// TIA Portal V16 export
// export: Created 2022-11-14T17:35:17.0009198Z, ExportSetting WithDefaults, DisplayName Totally Integrated Automation Portal, DisplayVersion V16, DisplayName TIA Portal Version Control Interface, DisplayVersion V16, DisplayName TIA Portal Openness, DisplayVersion V16, DisplayName STEP 7 Professional, DisplayVersion V16, DisplayName STEP 7 Safety, DisplayVersion V16, DisplayName WinCC Advanced, DisplayVersion V16
FUNCTION "FC03_TechnoplatAux" : Void   // FC3, LAD
TITLE = Auxiliary memory for the machine
{ S7_Optimized_Access := 'FALSE' }
AUTHOR : Robopac
VERSION : 0.0
// stored: AutoNumber false, IsIECCheckEnabled false, SetENOAutomatically false, UDAEnableTagReadback false
   VAR_INPUT
      PHASE : Bool;
   END_VAR
   VAR_TEMP
      Pulse_Reset : Bool;   // Pulse to reset encoders
      SuppSpeed : DWord;
      TempInt_min : Int;
      TempInt_max : Int;
      TempDint : DInt;
   END_VAR
   VAR_TEMP   // added for the SCL form of the ladder/FBD networks
      _w1 : Bool;
      _w2 : Bool;
      _w3 : Bool;
      _w4 : Bool;
   END_VAR
BEGIN

REGION Network 1: OSR and OSF for table phases sensor
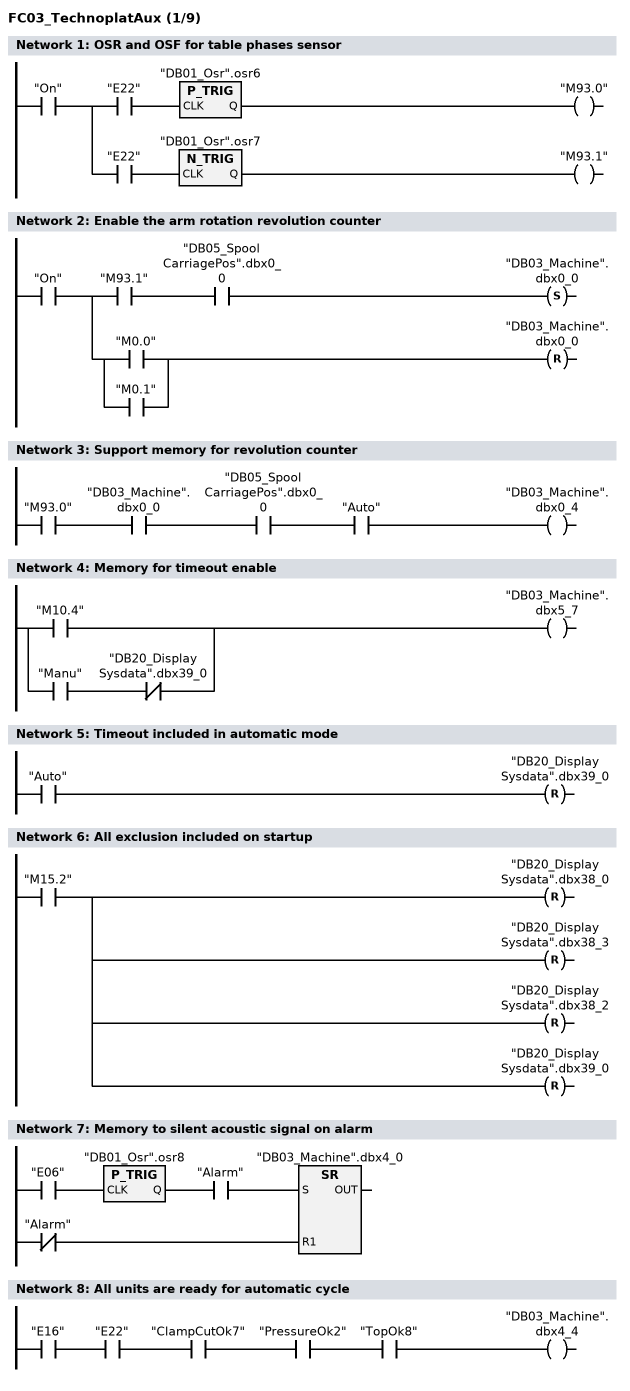
   RUNG wire#powerrail
      Contact( "On" )
      wire#w1
      Contact( "E22" )
      P_Trig( "DB01_Osr".osr6 )
      Coil( "M93.0" )
   END_RUNG
   RUNG wire#w1
      Contact( "E22" )
      N_Trig( "DB01_Osr".osr7 )
      Coil( "M93.1" )
   END_RUNG
   // the same network as SCL:
   #_w1 := "On" AND "E22";
   #_w2 := #_w1 AND NOT "DB01_Osr".osr6;   // rising edge
   "DB01_Osr".osr6 := #_w1;
   "M93.0" := #_w2;
   #_w3 := "On" AND "E22";
   #_w4 := NOT #_w3 AND "DB01_Osr".osr7;   // falling edge
   "DB01_Osr".osr7 := #_w3;
   "M93.1" := #_w4;
END_REGION

REGION Network 2: Enable the arm rotation revolution counter
   RUNG wire#powerrail
      Contact( "On" )
      wire#w1
      Contact( "M93.1" )
      Contact( "DB05_SpoolCarriagePos".dbx0_0 )
      S_Coil( "DB03_Machine".dbx0_0 )
   END_RUNG
   RUNG wire#w1
      Contact( "M0.0" )
      wire#w2
      R_Coil( "DB03_Machine".dbx0_0 )
   END_RUNG
   RUNG wire#w1
      Contact( "M0.1" )
   END_RUNG wire#w2
   // the same network as SCL:
   IF "On" AND "M93.1" AND "DB05_SpoolCarriagePos".dbx0_0 THEN "DB03_Machine".dbx0_0 := TRUE; END_IF;
   IF "On" AND ("M0.0" OR "M0.1") THEN "DB03_Machine".dbx0_0 := FALSE; END_IF;
END_REGION

REGION Network 3: Support memory for revolution counter
   RUNG wire#powerrail
      Contact( "M93.0" )
      Contact( "DB03_Machine".dbx0_0 )
      Contact( "DB05_SpoolCarriagePos".dbx0_0 )
      Contact( "Auto" )
      Coil( "DB03_Machine".dbx0_4 )
   END_RUNG
   // the same network as SCL:
   "DB03_Machine".dbx0_4 := "M93.0" AND "DB03_Machine".dbx0_0 AND "DB05_SpoolCarriagePos".dbx0_0 AND "Auto";
END_REGION

REGION Network 4: Memory for timeout enable
   RUNG wire#powerrail
      Contact( "M10.4" )
      wire#w1
      Coil( "DB03_Machine".dbx5_7 )
   END_RUNG
   RUNG wire#powerrail
      Contact( "Manu" )
      I_Contact( "DB20_DisplaySysdata".dbx39_0 )
   END_RUNG wire#w1
   // the same network as SCL:
   "DB03_Machine".dbx5_7 := "M10.4" OR ("Manu" AND NOT "DB20_DisplaySysdata".dbx39_0);
END_REGION

REGION Network 5: Timeout included in automatic mode
   RUNG wire#powerrail
      Contact( "Auto" )
      R_Coil( "DB20_DisplaySysdata".dbx39_0 )
   END_RUNG
   // the same network as SCL:
   IF "Auto" THEN "DB20_DisplaySysdata".dbx39_0 := FALSE; END_IF;
END_REGION

REGION Network 6: All exclusion included on startup
   RUNG wire#powerrail
      Contact( "M15.2" )
      wire#w1
      R_Coil( "DB20_DisplaySysdata".dbx38_0 )
   END_RUNG
   RUNG wire#w1
      R_Coil( "DB20_DisplaySysdata".dbx38_3 )
   END_RUNG
   RUNG wire#w1
      R_Coil( "DB20_DisplaySysdata".dbx38_2 )
   END_RUNG
   RUNG wire#w1
      R_Coil( "DB20_DisplaySysdata".dbx39_0 )
   END_RUNG
   // the same network as SCL:
   IF "M15.2" THEN
       "DB20_DisplaySysdata".dbx38_0 := FALSE;
       "DB20_DisplaySysdata".dbx38_3 := FALSE;
       "DB20_DisplaySysdata".dbx38_2 := FALSE;
       "DB20_DisplaySysdata".dbx39_0 := FALSE;
   END_IF;
END_REGION

REGION Network 7: Memory to silent acoustic signal on alarm
   RUNG wire#powerrail
      Contact( "E06" )
      P_Trig( "DB01_Osr".osr8 )
      Contact( "Alarm" )
      S_SR(operand := "DB03_Machine".dbx4_0, r1 := wire#w1)
   END_RUNG
   RUNG wire#powerrail
      I_Contact( "Alarm" )
   END_RUNG wire#w1
   // the same network as SCL:
   #_w1 := "E06" AND NOT "DB01_Osr".osr8;   // rising edge
   "DB01_Osr".osr8 := "E06";
   IF #_w1 AND "Alarm" THEN
       "DB03_Machine".dbx4_0 := TRUE;   // SR flip-flop
   END_IF;
   IF NOT "Alarm" THEN "DB03_Machine".dbx4_0 := FALSE; END_IF;
END_REGION

REGION Network 8: All units are ready for automatic cycle
   RUNG wire#powerrail
      Contact( "E16" )
      Contact( "E22" )
      Contact( "ClampCutOk7" )
      Contact( "PressureOk2" )
      Contact( "TopOk8" )
      Coil( "DB03_Machine".dbx4_4 )
   END_RUNG
   // the same network as SCL:
   "DB03_Machine".dbx4_4 := "E16" AND "E22" AND "ClampCutOk7" AND "PressureOk2" AND "TopOk8";
END_REGION

REGION Network 9: Prearrangement automatic cycle
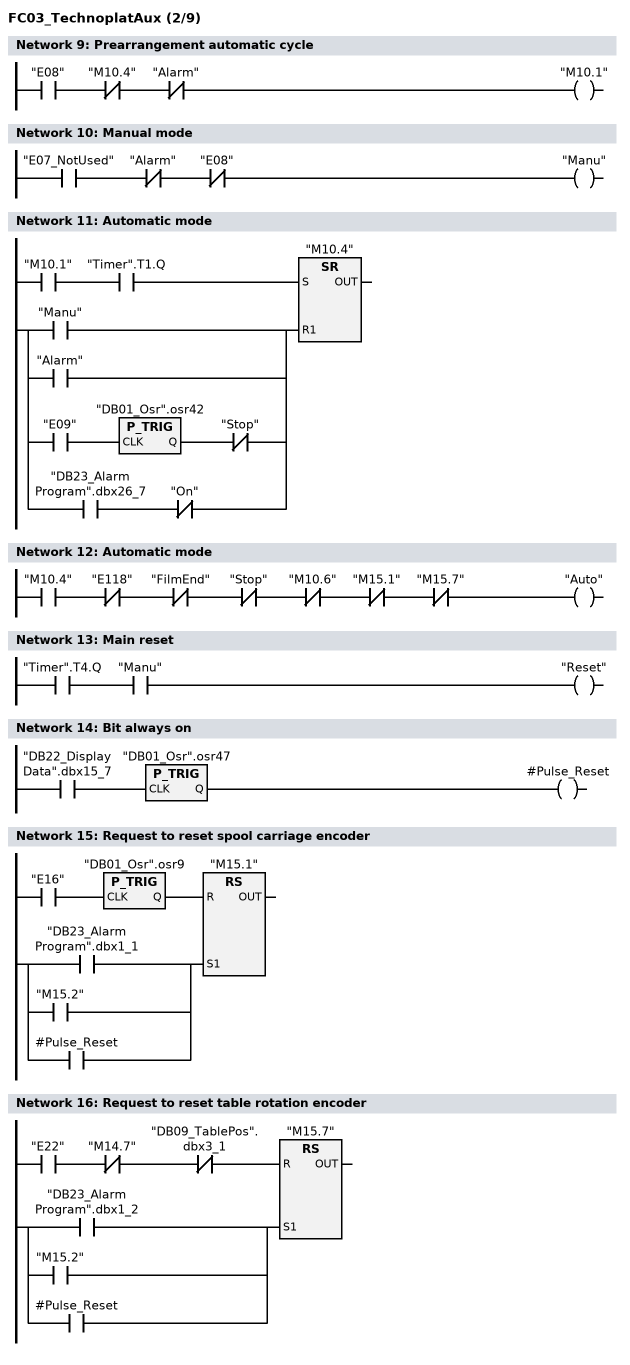
   RUNG wire#powerrail
      Contact( "E08" )
      I_Contact( "M10.4" )
      I_Contact( "Alarm" )
      Coil( "M10.1" )
   END_RUNG
   // the same network as SCL:
   "M10.1" := "E08" AND NOT "M10.4" AND NOT "Alarm";
END_REGION

REGION Network 10: Manual mode
   RUNG wire#powerrail
      Contact( "E07_NotUsed" )
      I_Contact( "Alarm" )
      I_Contact( "E08" )
      Coil( "Manu" )
   END_RUNG
   // the same network as SCL:
   "Manu" := "E07_NotUsed" AND NOT "Alarm" AND NOT "E08";
END_REGION

REGION Network 11: Automatic mode
   RUNG wire#powerrail
      Contact( "M10.1" )
      Contact( "Timer".T1.Q )
      S_SR(operand := "M10.4", r1 := wire#w1)
   END_RUNG
   RUNG wire#powerrail
      Contact( "Manu" )
   END_RUNG wire#w1
   RUNG wire#powerrail
      Contact( "Alarm" )
   END_RUNG wire#w1
   RUNG wire#powerrail
      Contact( "E09" )
      P_Trig( "DB01_Osr".osr42 )
      I_Contact( "Stop" )
   END_RUNG wire#w1
   RUNG wire#powerrail
      Contact( "DB23_AlarmProgram".dbx26_7 )
      I_Contact( "On" )
   END_RUNG wire#w1
   // the same network as SCL:
   #_w1 := "E09" AND NOT "DB01_Osr".osr42;   // rising edge
   "DB01_Osr".osr42 := "E09";
   IF "M10.1" AND "Timer".T1.Q THEN
       "M10.4" := TRUE;   // SR flip-flop
   END_IF;
   IF "Manu" OR "Alarm" OR (#_w1 AND NOT "Stop") OR ("DB23_AlarmProgram".dbx26_7 AND NOT "On") THEN
       "M10.4" := FALSE;
   END_IF;
END_REGION

REGION Network 12: Automatic mode
   RUNG wire#powerrail
      Contact( "M10.4" )
      I_Contact( "E118" )
      I_Contact( "FilmEnd" )
      I_Contact( "Stop" )
      I_Contact( "M10.6" )
      I_Contact( "M15.1" )
      I_Contact( "M15.7" )
      Coil( "Auto" )
   END_RUNG
   // the same network as SCL:
   "Auto" := "M10.4" AND NOT "E118" AND NOT "FilmEnd" AND NOT "Stop" AND NOT "M10.6" AND NOT "M15.1" AND NOT "M15.7";
END_REGION

REGION Network 13: Main reset
   RUNG wire#powerrail
      Contact( "Timer".T4.Q )
      Contact( "Manu" )
      Coil( "Reset" )
   END_RUNG
   // the same network as SCL:
   "Reset" := "Timer".T4.Q AND "Manu";
END_REGION

REGION Network 14: Bit always on
   RUNG wire#powerrail
      Contact( "DB22_DisplayData".dbx15_7 )
      P_Trig( "DB01_Osr".osr47 )
      Coil( #Pulse_Reset )
   END_RUNG
   // the same network as SCL:
   #_w1 := "DB22_DisplayData".dbx15_7 AND NOT "DB01_Osr".osr47;   // rising edge
   "DB01_Osr".osr47 := "DB22_DisplayData".dbx15_7;
   #Pulse_Reset := #_w1;
END_REGION

REGION Network 15: Request to reset spool carriage encoder
   RUNG wire#powerrail
      Contact( "E16" )
      P_Trig( "DB01_Osr".osr9 )
      S_RS(operand := "M15.1", s1 := wire#w1)
   END_RUNG
   RUNG wire#powerrail
      Contact( "DB23_AlarmProgram".dbx1_1 )
   END_RUNG wire#w1
   RUNG wire#powerrail
      Contact( "M15.2" )
   END_RUNG wire#w1
   RUNG wire#powerrail
      Contact( #Pulse_Reset )
   END_RUNG wire#w1
   // the same network as SCL:
   #_w1 := "E16" AND NOT "DB01_Osr".osr9;   // rising edge
   "DB01_Osr".osr9 := "E16";
   IF #_w1 THEN
       "M15.1" := FALSE;   // RS flip-flop
   END_IF;
   IF "DB23_AlarmProgram".dbx1_1 OR "M15.2" OR #Pulse_Reset THEN "M15.1" := TRUE; END_IF;
END_REGION

REGION Network 16: Request to reset table rotation encoder
   RUNG wire#powerrail
      Contact( "E22" )
      I_Contact( "M14.7" )
      I_Contact( "DB09_TablePos".dbx3_1 )
      S_RS(operand := "M15.7", s1 := wire#w1)
   END_RUNG
   RUNG wire#powerrail
      Contact( "DB23_AlarmProgram".dbx1_2 )
   END_RUNG wire#w1
   RUNG wire#powerrail
      Contact( "M15.2" )
   END_RUNG wire#w1
   RUNG wire#powerrail
      Contact( #Pulse_Reset )
   END_RUNG wire#w1
   // the same network as SCL:
   IF "E22" AND NOT "M14.7" AND NOT "DB09_TablePos".dbx3_1 THEN
       "M15.7" := FALSE;   // RS flip-flop
   END_IF;
   IF "DB23_AlarmProgram".dbx1_2 OR "M15.2" OR #Pulse_Reset THEN "M15.7" := TRUE; END_IF;
END_REGION

REGION Network 17: Table rotation backward to reset encoder
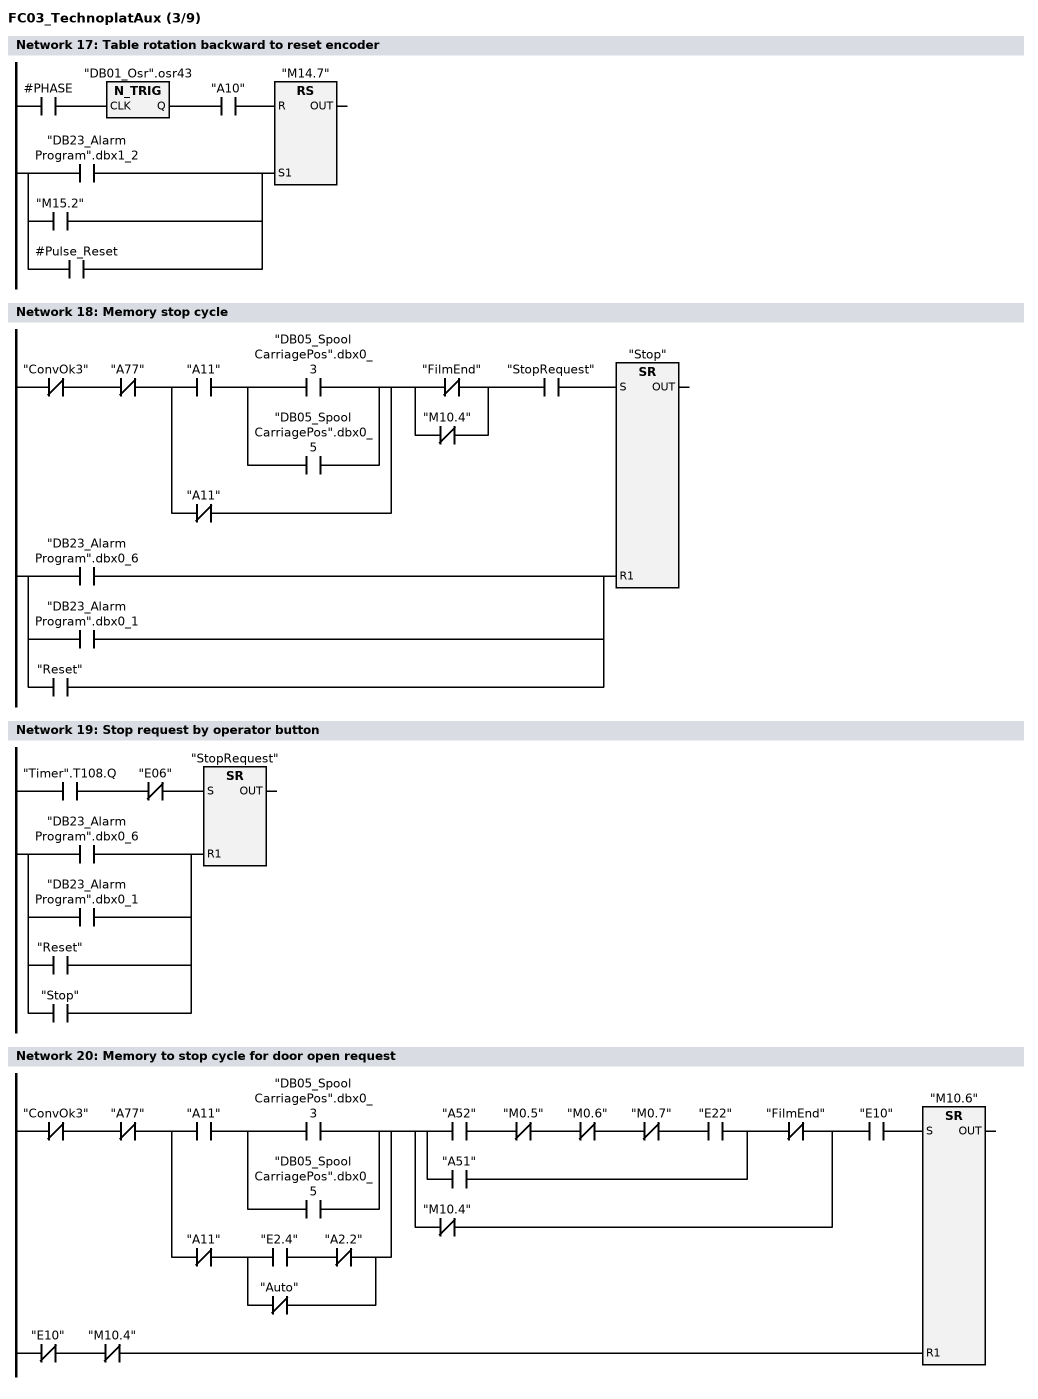
   RUNG wire#powerrail
      Contact( #PHASE )
      N_Trig( "DB01_Osr".osr43 )
      Contact( "A10" )
      S_RS(operand := "M14.7", s1 := wire#w1)
   END_RUNG
   RUNG wire#powerrail
      Contact( "DB23_AlarmProgram".dbx1_2 )
   END_RUNG wire#w1
   RUNG wire#powerrail
      Contact( "M15.2" )
   END_RUNG wire#w1
   RUNG wire#powerrail
      Contact( #Pulse_Reset )
   END_RUNG wire#w1
   // the same network as SCL:
   #_w1 := NOT #PHASE AND "DB01_Osr".osr43;   // falling edge
   "DB01_Osr".osr43 := #PHASE;
   IF #_w1 AND "A10" THEN
       "M14.7" := FALSE;   // RS flip-flop
   END_IF;
   IF "DB23_AlarmProgram".dbx1_2 OR "M15.2" OR #Pulse_Reset THEN "M14.7" := TRUE; END_IF;
END_REGION

REGION Network 18: Memory stop cycle
   RUNG wire#powerrail
      I_Contact( "ConvOk3" )
      I_Contact( "A77" )
      wire#w1
      Contact( "A11" )
      wire#w2
      Contact( "DB05_SpoolCarriagePos".dbx0_3 )
      wire#w3
      I_Contact( "FilmEnd" )
      wire#w4
      Contact( "StopRequest" )
      S_SR(operand := "Stop", r1 := wire#w5)
   END_RUNG
   RUNG wire#w2
      Contact( "DB05_SpoolCarriagePos".dbx0_5 )
   END_RUNG wire#w3
   RUNG wire#w1
      I_Contact( "A11" )
   END_RUNG wire#w3
   RUNG wire#w3
      I_Contact( "M10.4" )
   END_RUNG wire#w4
   RUNG wire#powerrail
      Contact( "DB23_AlarmProgram".dbx0_6 )
   END_RUNG wire#w5
   RUNG wire#powerrail
      Contact( "DB23_AlarmProgram".dbx0_1 )
   END_RUNG wire#w5
   RUNG wire#powerrail
      Contact( "Reset" )
   END_RUNG wire#w5
   // the same network as SCL:
   IF NOT "ConvOk3" AND NOT "A77" AND (("A11" AND ("DB05_SpoolCarriagePos".dbx0_3 OR "DB05_SpoolCarriagePos".dbx0_5)) OR NOT "A11") AND (NOT "FilmEnd" OR NOT "M10.4") AND "StopRequest" THEN
       "Stop" := TRUE;   // SR flip-flop
   END_IF;
   IF "DB23_AlarmProgram".dbx0_6 OR "DB23_AlarmProgram".dbx0_1 OR "Reset" THEN "Stop" := FALSE; END_IF;
END_REGION

REGION Network 19: Stop request by operator button
   RUNG wire#powerrail
      Contact( "Timer".T108.Q )
      I_Contact( "E06" )
      S_SR(operand := "StopRequest", r1 := wire#w1)
   END_RUNG
   RUNG wire#powerrail
      Contact( "DB23_AlarmProgram".dbx0_6 )
   END_RUNG wire#w1
   RUNG wire#powerrail
      Contact( "DB23_AlarmProgram".dbx0_1 )
   END_RUNG wire#w1
   RUNG wire#powerrail
      Contact( "Reset" )
   END_RUNG wire#w1
   RUNG wire#powerrail
      Contact( "Stop" )
   END_RUNG wire#w1
   // the same network as SCL:
   IF "Timer".T108.Q AND NOT "E06" THEN
       "StopRequest" := TRUE;   // SR flip-flop
   END_IF;
   IF "DB23_AlarmProgram".dbx0_6 OR "DB23_AlarmProgram".dbx0_1 OR "Reset" OR "Stop" THEN
       "StopRequest" := FALSE;
   END_IF;
END_REGION

REGION Network 20: Memory to stop cycle for door open request
   RUNG wire#powerrail
      I_Contact( "ConvOk3" )
      I_Contact( "A77" )
      wire#w1
      Contact( "A11" )
      wire#w2
      Contact( "DB05_SpoolCarriagePos".dbx0_3 )
      wire#w3
      Contact( "A52" )
      I_Contact( "M0.5" )
      I_Contact( "M0.6" )
      I_Contact( "M0.7" )
      Contact( "E22" )
      wire#w5
      I_Contact( "FilmEnd" )
      wire#w6
      Contact( "E10" )
      S_SR(operand := "M10.6", r1 := wire#w7)
   END_RUNG
   RUNG wire#w2
      Contact( "DB05_SpoolCarriagePos".dbx0_5 )
   END_RUNG wire#w3
   RUNG wire#w1
      I_Contact( "A11" )
      wire#w4
      Contact( "E2.4" )
      I_Contact( "A2.2" )
   END_RUNG wire#w3
   RUNG wire#w4
      I_Contact( "Auto" )
   END_RUNG wire#w3
   RUNG wire#w3
      Contact( "A51" )
   END_RUNG wire#w5
   RUNG wire#w3
      I_Contact( "M10.4" )
   END_RUNG wire#w6
   RUNG wire#powerrail
      I_Contact( "E10" )
      I_Contact( "M10.4" )
   END_RUNG wire#w7
   // the same network as SCL:
   IF NOT "ConvOk3" AND NOT "A77" AND (("A11" AND ("DB05_SpoolCarriagePos".dbx0_3 OR "DB05_SpoolCarriagePos".dbx0_5)) OR (NOT "A11" AND (("E2.4" AND NOT "A2.2") OR NOT "Auto"))) AND (((("A52" AND NOT "M0.5" AND NOT "M0.6" AND NOT "M0.7" AND "E22") OR "A51") AND NOT "FilmEnd") OR NOT "M10.4") AND "E10" THEN
       "M10.6" := TRUE;   // SR flip-flop
   END_IF;
   IF NOT "E10" AND NOT "M10.4" THEN "M10.6" := FALSE; END_IF;
END_REGION

REGION Network 21: Condition to check all out of positon alarm
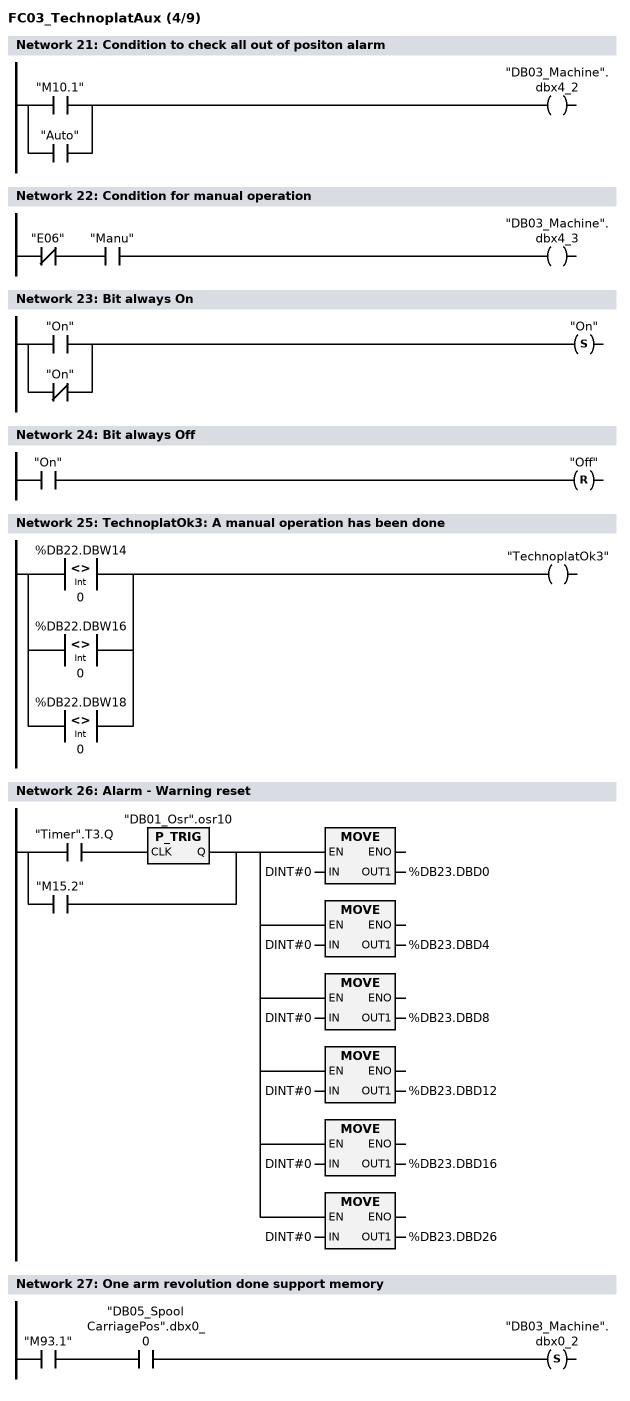
   RUNG wire#powerrail
      Contact( "M10.1" )
      wire#w1
      Coil( "DB03_Machine".dbx4_2 )
   END_RUNG
   RUNG wire#powerrail
      Contact( "Auto" )
   END_RUNG wire#w1
   // the same network as SCL:
   "DB03_Machine".dbx4_2 := "M10.1" OR "Auto";
END_REGION

REGION Network 22: Condition for manual operation
   RUNG wire#powerrail
      I_Contact( "E06" )
      Contact( "Manu" )
      Coil( "DB03_Machine".dbx4_3 )
   END_RUNG
   // the same network as SCL:
   "DB03_Machine".dbx4_3 := NOT "E06" AND "Manu";
END_REGION

REGION Network 23: Bit always On
   RUNG wire#powerrail
      Contact( "On" )
      wire#w1
      S_Coil( "On" )
   END_RUNG
   RUNG wire#powerrail
      I_Contact( "On" )
   END_RUNG wire#w1
   // the same network as SCL:
   IF "On" OR NOT "On" THEN "On" := TRUE; END_IF;
END_REGION

REGION Network 24: Bit always Off
   RUNG wire#powerrail
      Contact( "On" )
      R_Coil( "Off" )
   END_RUNG
   // the same network as SCL:
   IF "On" THEN "Off" := FALSE; END_IF;
END_REGION

REGION Network 25: TechnoplatOk3: A manual operation has been done
   RUNG wire#powerrail
      { S7_Templates := "SrcType := Int" } NE_Contact(in1 := %DB22.DBW14, in2 := 0)
      wire#w1
      Coil( "TechnoplatOk3" )
   END_RUNG
   RUNG wire#powerrail
      { S7_Templates := "SrcType := Int" } NE_Contact(in1 := %DB22.DBW16, in2 := 0)
   END_RUNG wire#w1
   RUNG wire#powerrail
      { S7_Templates := "SrcType := Int" } NE_Contact(in1 := %DB22.DBW18, in2 := 0)
   END_RUNG wire#w1
   // the same network as SCL:
   "TechnoplatOk3" := (%DB22.DBW14 <> 0) OR (%DB22.DBW16 <> 0) OR (%DB22.DBW18 <> 0);
END_REGION

REGION Network 26: Alarm - Warning reset
   RUNG wire#powerrail
      Contact( "Timer".T3.Q )
      P_Trig( "DB01_Osr".osr10 )
      wire#w1
      { S7_GenerateENO := "TRUE" } Move(in := DINT#0, out1 => %DB23.DBD0)
   END_RUNG
   RUNG wire#powerrail
      Contact( "M15.2" )
   END_RUNG wire#w1
   RUNG wire#w1
      { S7_GenerateENO := "TRUE" } Move(in := DINT#0, out1 => %DB23.DBD4)
   END_RUNG
   RUNG wire#w1
      { S7_GenerateENO := "TRUE" } Move(in := DINT#0, out1 => %DB23.DBD8)
   END_RUNG
   RUNG wire#w1
      { S7_GenerateENO := "TRUE" } Move(in := DINT#0, out1 => %DB23.DBD12)
   END_RUNG
   RUNG wire#w1
      { S7_GenerateENO := "TRUE" } Move(in := DINT#0, out1 => %DB23.DBD16)
   END_RUNG
   RUNG wire#w1
      { S7_GenerateENO := "TRUE" } Move(in := DINT#0, out1 => %DB23.DBD26)
   END_RUNG
   // the same network as SCL:
   #_w1 := "Timer".T3.Q AND NOT "DB01_Osr".osr10;   // rising edge
   "DB01_Osr".osr10 := "Timer".T3.Q;
   IF #_w1 OR "M15.2" THEN
       %DB23.DBD0 := DINT#0;
       %DB23.DBD4 := DINT#0;
       %DB23.DBD8 := DINT#0;
       %DB23.DBD12 := DINT#0;
       %DB23.DBD16 := DINT#0;
       %DB23.DBD26 := DINT#0;
   END_IF;
END_REGION

REGION Network 27: One arm revolution done support memory
   RUNG wire#powerrail
      Contact( "M93.1" )
      Contact( "DB05_SpoolCarriagePos".dbx0_0 )
      S_Coil( "DB03_Machine".dbx0_2 )
   END_RUNG
   // the same network as SCL:
   IF "M93.1" AND "DB05_SpoolCarriagePos".dbx0_0 THEN "DB03_Machine".dbx0_2 := TRUE; END_IF;
END_REGION

REGION Network 28: One arm revolution done
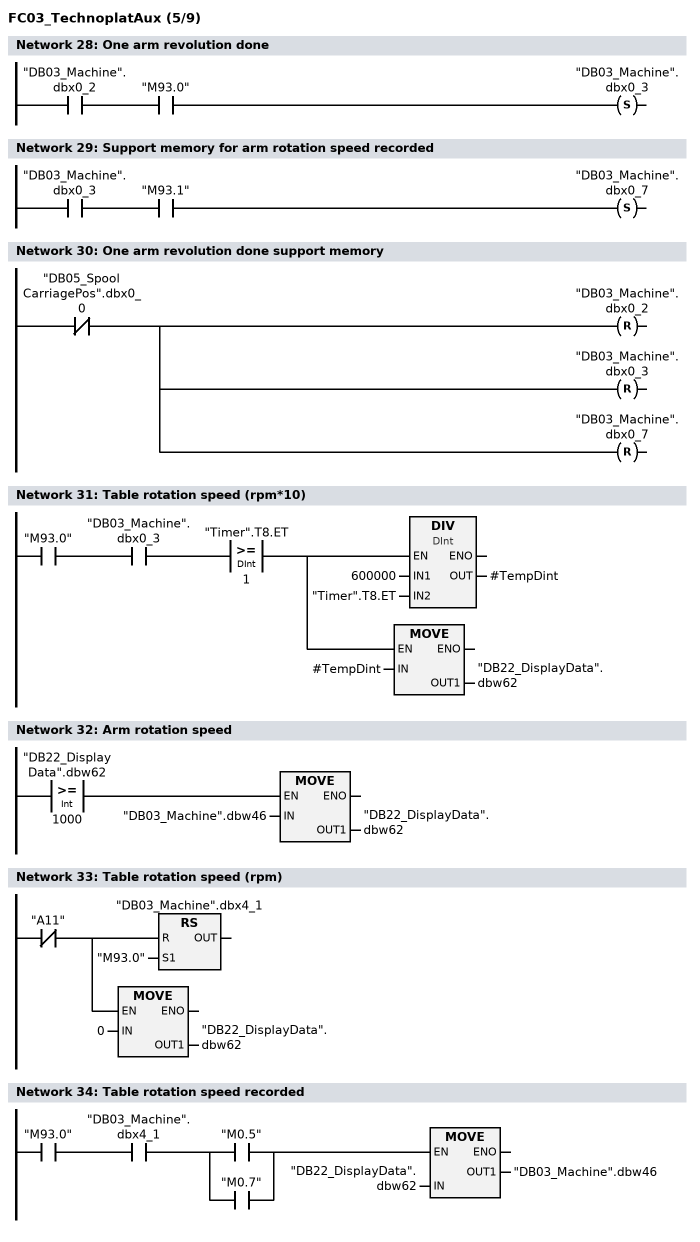
   RUNG wire#powerrail
      Contact( "DB03_Machine".dbx0_2 )
      Contact( "M93.0" )
      S_Coil( "DB03_Machine".dbx0_3 )
   END_RUNG
   // the same network as SCL:
   IF "DB03_Machine".dbx0_2 AND "M93.0" THEN "DB03_Machine".dbx0_3 := TRUE; END_IF;
END_REGION

REGION Network 29: Support memory for arm rotation speed recorded
   RUNG wire#powerrail
      Contact( "DB03_Machine".dbx0_3 )
      Contact( "M93.1" )
      S_Coil( "DB03_Machine".dbx0_7 )
   END_RUNG
   // the same network as SCL:
   IF "DB03_Machine".dbx0_3 AND "M93.1" THEN "DB03_Machine".dbx0_7 := TRUE; END_IF;
END_REGION

REGION Network 30: One arm revolution done support memory
   RUNG wire#powerrail
      I_Contact( "DB05_SpoolCarriagePos".dbx0_0 )
      wire#w1
      R_Coil( "DB03_Machine".dbx0_2 )
   END_RUNG
   RUNG wire#w1
      R_Coil( "DB03_Machine".dbx0_3 )
   END_RUNG
   RUNG wire#w1
      R_Coil( "DB03_Machine".dbx0_7 )
   END_RUNG
   // the same network as SCL:
   IF NOT "DB05_SpoolCarriagePos".dbx0_0 THEN
       "DB03_Machine".dbx0_2 := FALSE;
       "DB03_Machine".dbx0_3 := FALSE;
       "DB03_Machine".dbx0_7 := FALSE;
   END_IF;
END_REGION

REGION Network 31: Table rotation speed (rpm*10)
   RUNG wire#powerrail
      Contact( "M93.0" )
      Contact( "DB03_Machine".dbx0_3 )
      { S7_Templates := "SrcType := DInt" } GE_Contact(in1 := "Timer".T8.ET, in2 := 1)
      wire#w1
      { S7_Templates := "SrcType := DInt"; S7_GenerateENO := "TRUE" } Div(in1 := 600000, in2 := "Timer".T8.ET, out => #TempDint)
   END_RUNG
   RUNG wire#w1
      { S7_GenerateENO := "TRUE" } Move(in := #TempDint, out1 => "DB22_DisplayData".dbw62)
   END_RUNG
   // the same network as SCL:
   IF "M93.0" AND "DB03_Machine".dbx0_3 AND ("Timer".T8.ET >= 1) THEN
       #TempDint := 600000 / "Timer".T8.ET;
       "DB22_DisplayData".dbw62 := #TempDint;
   END_IF;
END_REGION

REGION Network 32: Arm rotation speed
   RUNG wire#powerrail
      { S7_Templates := "SrcType := Int" } GE_Contact(in1 := "DB22_DisplayData".dbw62, in2 := 1000)
      { S7_GenerateENO := "TRUE" } Move(in := "DB03_Machine".dbw46, out1 => "DB22_DisplayData".dbw62)
   END_RUNG
   // the same network as SCL:
   IF "DB22_DisplayData".dbw62 >= 1000 THEN "DB22_DisplayData".dbw62 := "DB03_Machine".dbw46; END_IF;
END_REGION

REGION Network 33: Table rotation speed (rpm)
   RUNG wire#powerrail
      I_Contact( "A11" )
      wire#w1
      S_RS(operand := "DB03_Machine".dbx4_1, s1 := "M93.0")
   END_RUNG
   RUNG wire#w1
      { S7_GenerateENO := "TRUE" } Move(in := 0, out1 => "DB22_DisplayData".dbw62)
   END_RUNG
   // the same network as SCL:
   IF NOT "A11" THEN
       "DB03_Machine".dbx4_1 := FALSE;   // RS flip-flop
   END_IF;
   IF "M93.0" THEN "DB03_Machine".dbx4_1 := TRUE; END_IF;
   IF NOT "A11" THEN "DB22_DisplayData".dbw62 := 0; END_IF;
END_REGION

REGION Network 34: Table rotation speed recorded
   RUNG wire#powerrail
      Contact( "M93.0" )
      Contact( "DB03_Machine".dbx4_1 )
      wire#w1
      Contact( "M0.5" )
      wire#w2
      { S7_GenerateENO := "TRUE" } Move(in := "DB22_DisplayData".dbw62, out1 => "DB03_Machine".dbw46)
   END_RUNG
   RUNG wire#w1
      Contact( "M0.7" )
   END_RUNG wire#w2
   // the same network as SCL:
   IF "M93.0" AND "DB03_Machine".dbx4_1 AND ("M0.5" OR "M0.7") THEN
       "DB03_Machine".dbw46 := "DB22_DisplayData".dbw62;
   END_IF;
END_REGION

REGION Network 35: Table rotation speed
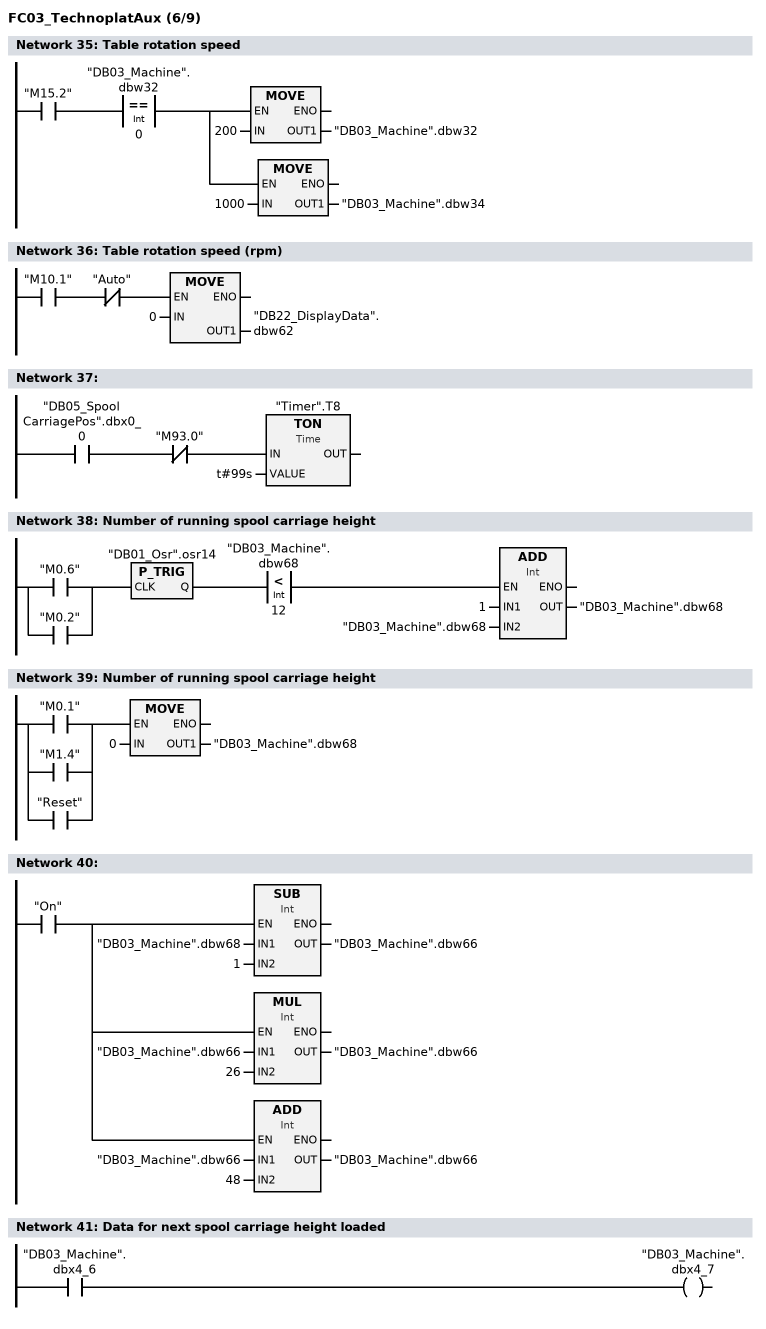
   RUNG wire#powerrail
      Contact( "M15.2" )
      { S7_Templates := "SrcType := Int" } EQ_Contact(in1 := "DB03_Machine".dbw32, in2 := 0)
      wire#w1
      { S7_GenerateENO := "TRUE" } Move(in := 200, out1 => "DB03_Machine".dbw32)
   END_RUNG
   RUNG wire#w1
      { S7_GenerateENO := "TRUE" } Move(in := 1000, out1 => "DB03_Machine".dbw34)
   END_RUNG
   // the same network as SCL:
   #_w1 := "M15.2" AND ("DB03_Machine".dbw32 = 0);
   IF #_w1 THEN
       "DB03_Machine".dbw32 := 200;
       "DB03_Machine".dbw34 := 1000;
   END_IF;
END_REGION

REGION Network 36: Table rotation speed (rpm)
   RUNG wire#powerrail
      Contact( "M10.1" )
      I_Contact( "Auto" )
      { S7_GenerateENO := "TRUE" } Move(in := 0, out1 => "DB22_DisplayData".dbw62)
   END_RUNG
   // the same network as SCL:
   IF "M10.1" AND NOT "Auto" THEN "DB22_DisplayData".dbw62 := 0; END_IF;
END_REGION

REGION Network 37
   "Timer".T8.TON(IN := "DB05_SpoolCarriagePos".dbx0_0 AND NOT "M93.0", PT := t#99s);   // TON coil
END_REGION

REGION Network 38: Number of running spool carriage height
   RUNG wire#powerrail
      Contact( "M0.6" )
      wire#w1
      P_Trig( "DB01_Osr".osr14 )
      { S7_Templates := "SrcType := Int" } LT_Contact(in1 := "DB03_Machine".dbw68, in2 := 12)
      { S7_Templates := "SrcType := Int"; S7_GenerateENO := "TRUE" } Add(in1 := 1, in2 := "DB03_Machine".dbw68, out => "DB03_Machine".dbw68)
   END_RUNG
   RUNG wire#powerrail
      Contact( "M0.2" )
   END_RUNG wire#w1
   // the same network as SCL:
   #_w1 := "M0.6" OR "M0.2";
   #_w2 := #_w1 AND NOT "DB01_Osr".osr14;   // rising edge
   "DB01_Osr".osr14 := #_w1;
   IF #_w2 AND ("DB03_Machine".dbw68 < 12) THEN "DB03_Machine".dbw68 := 1 + "DB03_Machine".dbw68; END_IF;
END_REGION

REGION Network 39: Number of running spool carriage height
   RUNG wire#powerrail
      Contact( "M0.1" )
      wire#w1
      { S7_GenerateENO := "TRUE" } Move(in := 0, out1 => "DB03_Machine".dbw68)
   END_RUNG
   RUNG wire#powerrail
      Contact( "M1.4" )
   END_RUNG wire#w1
   RUNG wire#powerrail
      Contact( "Reset" )
   END_RUNG wire#w1
   // the same network as SCL:
   IF "M0.1" OR "M1.4" OR "Reset" THEN "DB03_Machine".dbw68 := 0; END_IF;
END_REGION

REGION Network 40
   RUNG wire#powerrail
      Contact( "On" )
      wire#w1
      { S7_Templates := "SrcType := Int"; S7_GenerateENO := "TRUE" } Sub(in1 := "DB03_Machine".dbw68, in2 := 1, out => "DB03_Machine".dbw66)
   END_RUNG
   RUNG wire#w1
      { S7_Templates := "SrcType := Int"; S7_GenerateENO := "TRUE" } Mul(in1 := "DB03_Machine".dbw66, in2 := 26, out => "DB03_Machine".dbw66)
   END_RUNG
   RUNG wire#w1
      { S7_Templates := "SrcType := Int"; S7_GenerateENO := "TRUE" } Add(in1 := "DB03_Machine".dbw66, in2 := 48, out => "DB03_Machine".dbw66)
   END_RUNG
   // the same network as SCL:
   IF "On" THEN
       "DB03_Machine".dbw66 := "DB03_Machine".dbw68 - 1;
       "DB03_Machine".dbw66 := "DB03_Machine".dbw66 * 26;
       "DB03_Machine".dbw66 := "DB03_Machine".dbw66 + 48;
   END_IF;
END_REGION

REGION Network 41: Data for next spool carriage height loaded
   RUNG wire#powerrail
      Contact( "DB03_Machine".dbx4_6 )
      Coil( "DB03_Machine".dbx4_7 )
   END_RUNG
   // the same network as SCL:
   "DB03_Machine".dbx4_7 := "DB03_Machine".dbx4_6;
END_REGION

REGION Network 42: Moving data for the running quote
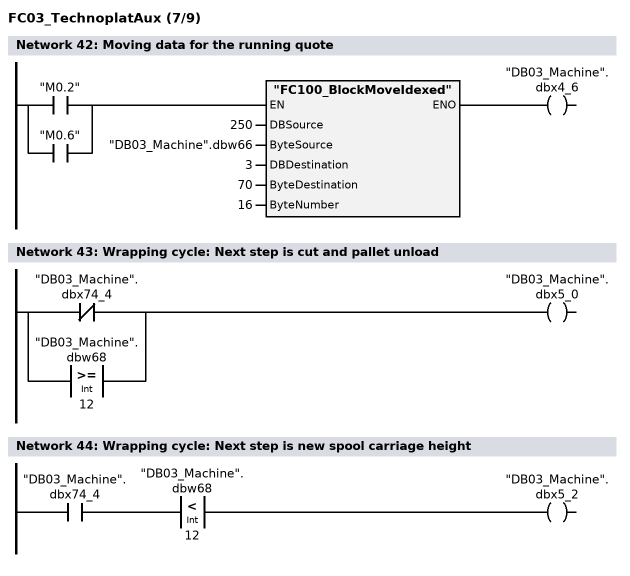
   RUNG wire#powerrail
      Contact( "M0.2" )
      wire#w1
      "FC100_BlockMoveIdexed"(DBSource := 250, ByteSource := "DB03_Machine".dbw66, DBDestination := 3, ByteDestination := 70, ByteNumber := 16)
      Coil( "DB03_Machine".dbx4_6 )
   END_RUNG
   RUNG wire#powerrail
      Contact( "M0.6" )
   END_RUNG wire#w1
   // the same network as SCL:
   "FC100_BlockMoveIdexed"(EN := "M0.2" OR "M0.6",
                           DBSource := 250,
                           ByteSource := "DB03_Machine".dbw66,
                           DBDestination := 3,
                           ByteDestination := 70,
                           ByteNumber := 16,
                           ENO => #_w1);
   "DB03_Machine".dbx4_6 := #_w1;
END_REGION

REGION Network 43: Wrapping cycle: Next step is cut and pallet unload
   RUNG wire#powerrail
      I_Contact( "DB03_Machine".dbx74_4 )
      wire#w1
      Coil( "DB03_Machine".dbx5_0 )
   END_RUNG
   RUNG wire#powerrail
      { S7_Templates := "SrcType := Int" } GE_Contact(in1 := "DB03_Machine".dbw68, in2 := 12)
   END_RUNG wire#w1
   // the same network as SCL:
   "DB03_Machine".dbx5_0 := NOT "DB03_Machine".dbx74_4 OR ("DB03_Machine".dbw68 >= 12);
END_REGION

REGION Network 44: Wrapping cycle: Next step is new spool carriage height
   RUNG wire#powerrail
      Contact( "DB03_Machine".dbx74_4 )
      { S7_Templates := "SrcType := Int" } LT_Contact(in1 := "DB03_Machine".dbw68, in2 := 12)
      Coil( "DB03_Machine".dbx5_2 )
   END_RUNG
   // the same network as SCL:
   "DB03_Machine".dbx5_2 := "DB03_Machine".dbx74_4 AND ("DB03_Machine".dbw68 < 12);
END_REGION

REGION Network 45: Wrong data program for the pallet on the machine
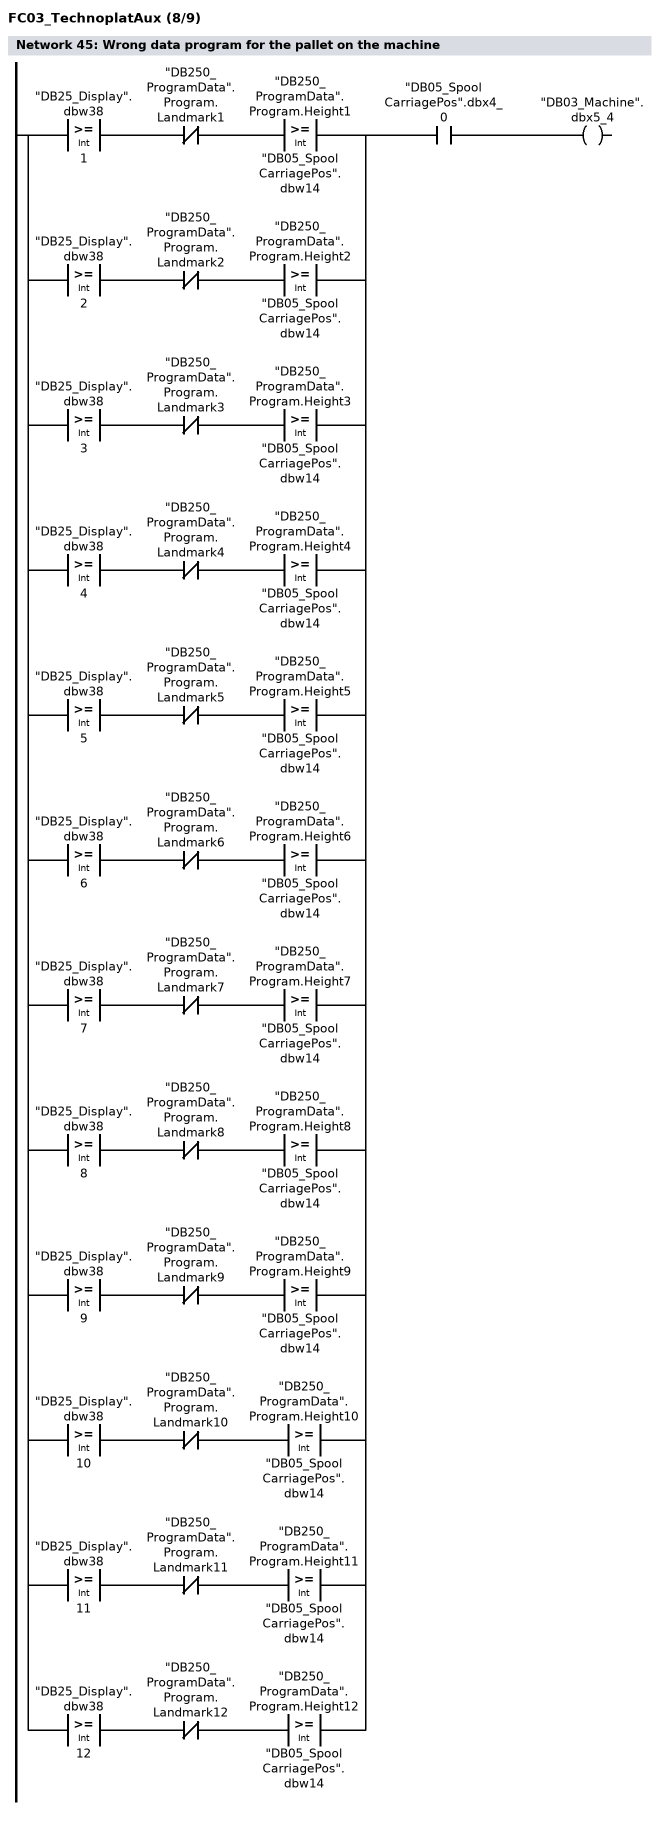
   RUNG wire#powerrail
      { S7_Templates := "SrcType := Int" } GE_Contact(in1 := "DB25_Display".dbw38, in2 := 1)
      I_Contact( "DB250_ProgramData".Program.Landmark1 )
      { S7_Templates := "SrcType := Int" } GE_Contact(in1 := "DB250_ProgramData".Program.Height1, in2 := "DB05_SpoolCarriagePos".dbw14)
      wire#w1
      Contact( "DB05_SpoolCarriagePos".dbx4_0 )
      Coil( "DB03_Machine".dbx5_4 )
   END_RUNG
   RUNG wire#powerrail
      { S7_Templates := "SrcType := Int" } GE_Contact(in1 := "DB25_Display".dbw38, in2 := 2)
      I_Contact( "DB250_ProgramData".Program.Landmark2 )
      { S7_Templates := "SrcType := Int" } GE_Contact(in1 := "DB250_ProgramData".Program.Height2, in2 := "DB05_SpoolCarriagePos".dbw14)
   END_RUNG wire#w1
   RUNG wire#powerrail
      { S7_Templates := "SrcType := Int" } GE_Contact(in1 := "DB25_Display".dbw38, in2 := 3)
      I_Contact( "DB250_ProgramData".Program.Landmark3 )
      { S7_Templates := "SrcType := Int" } GE_Contact(in1 := "DB250_ProgramData".Program.Height3, in2 := "DB05_SpoolCarriagePos".dbw14)
   END_RUNG wire#w1
   RUNG wire#powerrail
      { S7_Templates := "SrcType := Int" } GE_Contact(in1 := "DB25_Display".dbw38, in2 := 4)
      I_Contact( "DB250_ProgramData".Program.Landmark4 )
      { S7_Templates := "SrcType := Int" } GE_Contact(in1 := "DB250_ProgramData".Program.Height4, in2 := "DB05_SpoolCarriagePos".dbw14)
   END_RUNG wire#w1
   RUNG wire#powerrail
      { S7_Templates := "SrcType := Int" } GE_Contact(in1 := "DB25_Display".dbw38, in2 := 5)
      I_Contact( "DB250_ProgramData".Program.Landmark5 )
      { S7_Templates := "SrcType := Int" } GE_Contact(in1 := "DB250_ProgramData".Program.Height5, in2 := "DB05_SpoolCarriagePos".dbw14)
   END_RUNG wire#w1
   RUNG wire#powerrail
      { S7_Templates := "SrcType := Int" } GE_Contact(in1 := "DB25_Display".dbw38, in2 := 6)
      I_Contact( "DB250_ProgramData".Program.Landmark6 )
      { S7_Templates := "SrcType := Int" } GE_Contact(in1 := "DB250_ProgramData".Program.Height6, in2 := "DB05_SpoolCarriagePos".dbw14)
   END_RUNG wire#w1
   RUNG wire#powerrail
      { S7_Templates := "SrcType := Int" } GE_Contact(in1 := "DB25_Display".dbw38, in2 := 7)
      I_Contact( "DB250_ProgramData".Program.Landmark7 )
      { S7_Templates := "SrcType := Int" } GE_Contact(in1 := "DB250_ProgramData".Program.Height7, in2 := "DB05_SpoolCarriagePos".dbw14)
   END_RUNG wire#w1
   RUNG wire#powerrail
      { S7_Templates := "SrcType := Int" } GE_Contact(in1 := "DB25_Display".dbw38, in2 := 8)
      I_Contact( "DB250_ProgramData".Program.Landmark8 )
      { S7_Templates := "SrcType := Int" } GE_Contact(in1 := "DB250_ProgramData".Program.Height8, in2 := "DB05_SpoolCarriagePos".dbw14)
   END_RUNG wire#w1
   RUNG wire#powerrail
      { S7_Templates := "SrcType := Int" } GE_Contact(in1 := "DB25_Display".dbw38, in2 := 9)
      I_Contact( "DB250_ProgramData".Program.Landmark9 )
      { S7_Templates := "SrcType := Int" } GE_Contact(in1 := "DB250_ProgramData".Program.Height9, in2 := "DB05_SpoolCarriagePos".dbw14)
   END_RUNG wire#w1
   RUNG wire#powerrail
      { S7_Templates := "SrcType := Int" } GE_Contact(in1 := "DB25_Display".dbw38, in2 := 10)
      I_Contact( "DB250_ProgramData".Program.Landmark10 )
      { S7_Templates := "SrcType := Int" } GE_Contact(in1 := "DB250_ProgramData".Program.Height10, in2 := "DB05_SpoolCarriagePos".dbw14)
   END_RUNG wire#w1
   RUNG wire#powerrail
      { S7_Templates := "SrcType := Int" } GE_Contact(in1 := "DB25_Display".dbw38, in2 := 11)
      I_Contact( "DB250_ProgramData".Program.Landmark11 )
      { S7_Templates := "SrcType := Int" } GE_Contact(in1 := "DB250_ProgramData".Program.Height11, in2 := "DB05_SpoolCarriagePos".dbw14)
   END_RUNG wire#w1
   RUNG wire#powerrail
      { S7_Templates := "SrcType := Int" } GE_Contact(in1 := "DB25_Display".dbw38, in2 := 12)
      I_Contact( "DB250_ProgramData".Program.Landmark12 )
      { S7_Templates := "SrcType := Int" } GE_Contact(in1 := "DB250_ProgramData".Program.Height12, in2 := "DB05_SpoolCarriagePos".dbw14)
   END_RUNG wire#w1
   // the same network as SCL:
   "DB03_Machine".dbx5_4 := ((("DB25_Display".dbw38 >= 1) AND NOT "DB250_ProgramData".Program.Landmark1 AND ("DB250_ProgramData".Program.Height1 >= "DB05_SpoolCarriagePos".dbw14)) OR (("DB25_Display".dbw38 >= 2) AND NOT "DB250_ProgramData".Program.Landmark2 AND ("DB250_ProgramData".Program.Height2 >= "DB05_SpoolCarriagePos".dbw14)) OR (("DB25_Display".dbw38 >= 3) AND NOT "DB250_ProgramData".Program.Landmark3 AND ("DB250_ProgramData".Program.Height3 >= "DB05_SpoolCarriagePos".dbw14)) OR (("DB25_Display".dbw38 >= 4) AND NOT "DB250_ProgramData".Program.Landmark4 AND ("DB250_ProgramData".Program.Height4 >= "DB05_SpoolCarriagePos".dbw14)) OR (("DB25_Display".dbw38 >= 5) AND NOT "DB250_ProgramData".Program.Landmark5 AND ("DB250_ProgramData".Program.Height5 >= "DB05_SpoolCarriagePos".dbw14)) OR (("DB25_Display".dbw38 >= 6) AND NOT "DB250_ProgramData".Program.Landmark6 AND ("DB250_ProgramData".Program.Height6 >= "DB05_SpoolCarriagePos".dbw14)) OR (("DB25_Display".dbw38 >= 7) AND NOT "DB250_ProgramData".Program.Landmark7 AND ("DB250_ProgramData".Program.Height7 >= "DB05_SpoolCarriagePos".dbw14)) OR (("DB25_Display".dbw38 >= 8) AND NOT "DB250_ProgramData".Program.Landmark8 AND ("DB250_ProgramData".Program.Height8 >= "DB05_SpoolCarriagePos".dbw14)) OR (("DB25_Display".dbw38 >= 9) AND NOT "DB250_ProgramData".Program.Landmark9 AND ("DB250_ProgramData".Program.Height9 >= "DB05_SpoolCarriagePos".dbw14)) OR (("DB25_Display".dbw38 >= 10) AND NOT "DB250_ProgramData".Program.Landmark10 AND ("DB250_ProgramData".Program.Height10 >= "DB05_SpoolCarriagePos".dbw14)) OR (("DB25_Display".dbw38 >= 11) AND NOT "DB250_ProgramData".Program.Landmark11 AND ("DB250_ProgramData".Program.Height11 >= "DB05_SpoolCarriagePos".dbw14)) OR (("DB25_Display".dbw38 >= 12) AND NOT "DB250_ProgramData".Program.Landmark12 AND ("DB250_ProgramData".Program.Height12 >= "DB05_SpoolCarriagePos".dbw14))) AND "DB05_SpoolCarriagePos".dbx4_0;
END_REGION

REGION Network 46: Automatic mode for external conveyors
   // il transito tra 4 e 5 va sempre completato (in caso di richiesta E118 o porta non aperta /E119)
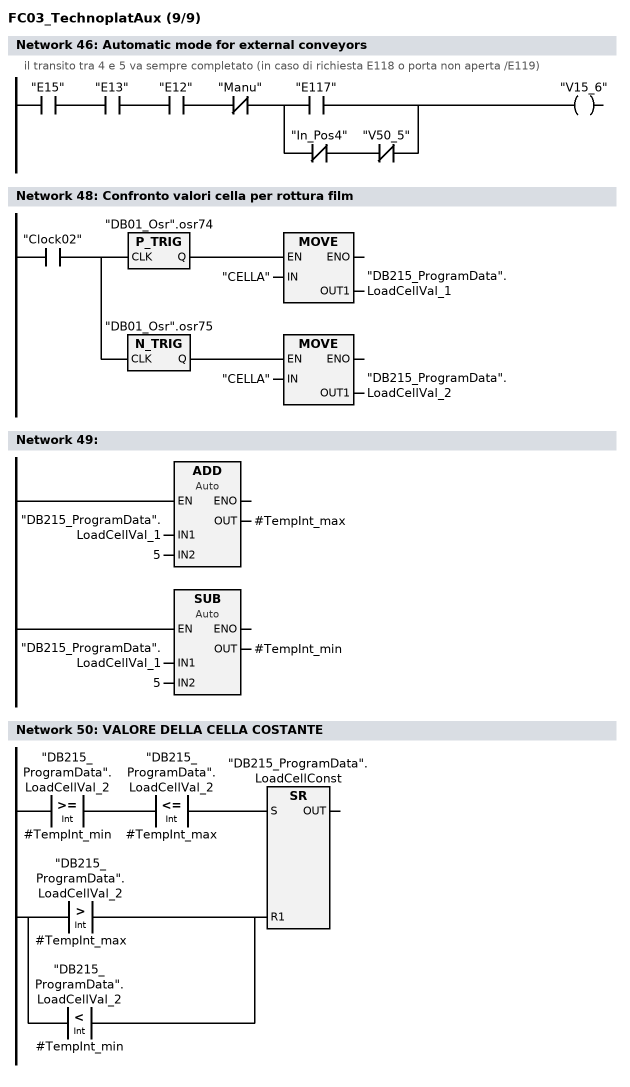
   RUNG wire#powerrail
      Contact( "E15" )
      Contact( "E13" )
      Contact( "E12" )
      I_Contact( "Manu" )
      wire#w1
      Contact( "E117" )
      wire#w2
      Coil( "V15_6" )
   END_RUNG
   RUNG wire#w1
      I_Contact( "In_Pos4" )
      I_Contact( "V50_5" )
   END_RUNG wire#w2
   // the same network as SCL:
   "V15_6" := "E15" AND "E13" AND "E12" AND NOT "Manu" AND ("E117" OR (NOT "In_Pos4" AND NOT "V50_5"));
END_REGION

REGION Network 47: ROTTURA FILM
END_REGION

REGION Network 48: Confronto valori cella per rottura film
   RUNG wire#powerrail
      Contact( "Clock02" )
      wire#w1
      P_Trig( "DB01_Osr".osr74 )
      Move(in := "CELLA", out1 => "DB215_ProgramData".LoadCellVal_1)
   END_RUNG
   RUNG wire#w1
      N_Trig( "DB01_Osr".osr75 )
      Move(in := "CELLA", out1 => "DB215_ProgramData".LoadCellVal_2)
   END_RUNG
   // the same network as SCL:
   #_w1 := "Clock02" AND NOT "DB01_Osr".osr74;   // rising edge
   "DB01_Osr".osr74 := "Clock02";
   IF #_w1 THEN "DB215_ProgramData".LoadCellVal_1 := "CELLA"; END_IF;
   #_w2 := NOT "Clock02" AND "DB01_Osr".osr75;   // falling edge
   "DB01_Osr".osr75 := "Clock02";
   IF #_w2 THEN "DB215_ProgramData".LoadCellVal_2 := "CELLA"; END_IF;
END_REGION

REGION Network 49
   RUNG wire#powerrail
      Add(in1 := "DB215_ProgramData".LoadCellVal_1, in2 := 5, out => #TempInt_max)
   END_RUNG
   RUNG wire#powerrail
      Sub(in1 := "DB215_ProgramData".LoadCellVal_1, in2 := 5, out => #TempInt_min)
   END_RUNG
   // the same network as SCL:
   #TempInt_max := "DB215_ProgramData".LoadCellVal_1 + 5;
   #TempInt_min := "DB215_ProgramData".LoadCellVal_1 - 5;
END_REGION

REGION Network 50: VALORE DELLA CELLA COSTANTE
   RUNG wire#powerrail
      { S7_Templates := "SrcType := Int" } GE_Contact(in1 := "DB215_ProgramData".LoadCellVal_2, in2 := #TempInt_min)
      { S7_Templates := "SrcType := Int" } LE_Contact(in1 := "DB215_ProgramData".LoadCellVal_2, in2 := #TempInt_max)
      S_SR(operand := "DB215_ProgramData".LoadCellConst, r1 := wire#w1)
   END_RUNG
   RUNG wire#powerrail
      { S7_Templates := "SrcType := Int" } GT_Contact(in1 := "DB215_ProgramData".LoadCellVal_2, in2 := #TempInt_max)
   END_RUNG wire#w1
   RUNG wire#powerrail
      { S7_Templates := "SrcType := Int" } LT_Contact(in1 := "DB215_ProgramData".LoadCellVal_2, in2 := #TempInt_min)
   END_RUNG wire#w1
   // the same network as SCL:
   IF ("DB215_ProgramData".LoadCellVal_2 >= #TempInt_min) AND ("DB215_ProgramData".LoadCellVal_2 <= #TempInt_max) THEN
       "DB215_ProgramData".LoadCellConst := TRUE;   // SR flip-flop
   END_IF;
   IF ("DB215_ProgramData".LoadCellVal_2 > #TempInt_max) OR ("DB215_ProgramData".LoadCellVal_2 < #TempInt_min) THEN
       "DB215_ProgramData".LoadCellConst := FALSE;
   END_IF;
END_REGION
END_FUNCTION
